{attribute 'hide'}
FUNCTION_BLOCK NullEntry_Test EXTENDS TcUnit.FB_TestSuite

IsNullReturnsExpected();

METHOD IsNullReturnsExpected
VAR
	result : BOOL;
	nullEntry : NullEntry('');
END_VAR
TEST('IsNullReturnsExpected');

// @TEST-FIXTURE

// @TEST-RUN
result := nullEntry.IsNull;

// @TEST-ASSSERT
AssertTrue(Condition := result, Message := 'IsNull did not return TRUE');

TEST_FINISHED();
END_METHOD

END_FUNCTION_BLOCK

(* stored: Version 1.1.0.1, ProductVersion 3.1.4024.9
   POU NullEntry_Test: Id {124b9b06-390b-49c4-b8ac-9fe7314e4452}, SpecialFunc None
   Method IsNullReturnsExpected: Id {b828288d-cdff-443d-a973-ef3aee41f7cd} *)
